FUNCTION F_AccDecDistanceFromVelo : LREAL
VAR_INPUT
	nVelocity	: LREAL ; // velocity [m/s]
	nAccDecc	: LREAL ; // acceleration or deceleration value [m/s^2]
END_VAR
VAR
	nTime : LREAL ;
END_VAR

nTime := nVelocity	/	nAccDecc ;

F_AccDecDistanceFromVelo := nVelocity * (nTime/2);

END_FUNCTION

(* stored: Version 1.1.0.1, ProductVersion 3.1.4024.3
   POU F_AccDecDistanceFromVelo: Id {0f2c97ac-1162-4662-90b2-4c9665676ae7}, SpecialFunc None *)
